(* IEC 61131-3 sources: Masterarbeit/sigmatek/lasalclass2/PW022_hardware/Class/Steuerung, 1 file *)

(* ---- Steuerung.st ---- *)
(*!
<Class
	Name               = "Steuerung"
	Revision           = "0.0"
	RealtimeTask       = "true"
	DefRealtime        = "1000 ms"
	CyclicTask         = "false"
	DefCyclictime      = "10 ms"
	BackgroundTask     = "false"
	Sigmatek           = "false"
	OSInterface        = "false"
	HighPriority       = "false"
	Automatic          = "false"
	UpdateMode         = "Prescan"
	SharedCommandTable = "true"
	Objectsize         = "(428,120)">
	<Channels>
		<Server Name="ClassSvr" Visualized="false" Initialize="false" WriteProtected="true" Retentive="false"/>
		<Server Name="Start" Visualized="false" Initialize="false" WriteProtected="false" Retentive="false"/>
		<Server Name="Stop" Visualized="false" Initialize="false" WriteProtected="false" Retentive="false"/>
		<Client Name="cPeriodeDuration_ch1" Required="true" Internal="false"/>
		<Client Name="cPeriodeDuration_ch2" Required="true" Internal="false"/>
		<Client Name="cPeriodeDuration_ch3" Required="true" Internal="false"/>
		<Client Name="cPeriodeDuration_ch4" Required="true" Internal="false"/>
		<Client Name="cPeriodeDuration_ch5" Required="true" Internal="false"/>
		<Client Name="cPeriodeDuration_ch6" Required="true" Internal="false"/>
		<Client Name="cPWMOnTime_ch1" Required="true" Internal="false"/>
		<Client Name="cPWMOnTime_ch2" Required="true" Internal="false"/>
		<Client Name="cPWMOnTime_ch3" Required="true" Internal="false"/>
		<Client Name="cPWMOnTime_ch4" Required="true" Internal="false"/>
		<Client Name="cPWMOnTime_ch5" Required="true" Internal="false"/>
		<Client Name="cPWMOnTime_ch6" Required="true" Internal="false"/>
	</Channels>
</Class>
*)
Steuerung : CLASS
  //Servers:
	ClassSvr 	: SvrChCmd_DINT;
	Stop 	: SvrCh_DINT;
	Start 	: SvrCh_DINT;
  //Clients:
	cPeriodeDuration_ch1 	: CltCh_DINT;
	cPWMOnTime_ch1 	: CltCh_DINT;
	cPeriodeDuration_ch2 	: CltCh_DINT;
	cPWMOnTime_ch2 	: CltCh_DINT;
	cPeriodeDuration_ch3 	: CltCh_DINT;
	cPWMOnTime_ch3 	: CltCh_DINT;
	cPeriodeDuration_ch4 	: CltCh_DINT;
	cPWMOnTime_ch4 	: CltCh_DINT;
	cPeriodeDuration_ch5 	: CltCh_DINT;
	cPWMOnTime_ch5 	: CltCh_DINT;
	cPeriodeDuration_ch6 	: CltCh_DINT;
	cPWMOnTime_ch6 	: CltCh_DINT;
  //Variables:
		Timemark1 	: UDINT;
		Timemark2 	: UDINT;
		AverageLatency_us 	: REAL;
		AverageLatency_ns 	: REAL;
		AverageLatency_raw 	: REAL;
  //Functions:

	FUNCTION VIRTUAL GLOBAL Init;

	FUNCTION VIRTUAL GLOBAL RtWork
		VAR_INPUT
			EAX 	: UDINT;
		END_VAR
		VAR_OUTPUT
			state (EAX) 	: UDINT;
		END_VAR;
  //Tables:
	FUNCTION @STD
		VAR_OUTPUT
			ret_code	: CONFSTATES;
		END_VAR;
	FUNCTION GLOBAL TAB @CT_;
END_CLASS;

FUNCTION VIRTUAL GLOBAL Steuerung::Init
    if _FirstScan = TRUE then
        cPeriodeDuration_ch1.Write(20000);
        cPeriodeDuration_ch2.Write(20000);
        cPeriodeDuration_ch3.Write(20000);
        cPeriodeDuration_ch4.Write(20000);
        cPeriodeDuration_ch5.Write(20000);
        cPeriodeDuration_ch6.Write(20000);
    end_if;
END_FUNCTION

FUNCTION VIRTUAL GLOBAL Steuerung::RtWork
    VAR_INPUT
        EAX : UDINT;
    END_VAR
    VAR_OUTPUT
        state (EAX) : UDINT;
    END_VAR
    VAR
  	  i : DINT;
    END_VAR

    // Record the start time
    Timemark1 := OS_READMICROSEC();

    // Loop to send commands and measure latency
    for i := 0 to 999 do
        cPWMOnTime_ch1.Write(100);
        cPWMOnTime_ch2.Write(200);
        cPWMOnTime_ch3.Write(300);
        cPWMOnTime_ch4.Write(400);
        cPWMOnTime_ch5.Write(500);
        cPWMOnTime_ch6.Write(600);
    end_for;

    // Record the end time
    Timemark2 := OS_READMICROSEC();

    // Calculate average latency per operation
    AverageLatency_raw := (Timemark2 - Timemark1);
    AverageLatency_us := AverageLatency_raw / 1000;
    AverageLatency_ns := AverageLatency_us * 1000;

    state := READY;
END_FUNCTION
